TYPE ST_Outputs :
STRUCT	
	GRIP_CLOSE				: BOOL;
	JOINT_TURN		  		: ARRAY [1..GVL_RobotArmConstants.MAX_NUMBER_OF_JOINTS] OF ST_JointDirection;
END_STRUCT
END_TYPE

(* stored: Version 1.1.0.1, ProductVersion 3.1.4024.9
   DUT ST_Outputs: Id {0304fd20-21e7-467d-aa49-8a654f790651} *)
